// TIA Portal V19 export
FUNCTION_BLOCK "F_Zone13_FB"   // FB184, F_LAD
TITLE = SAFETY ZONE 11 - AREA 02 (FINAL CUT)
// -
// stored: Access Published
   VAR
      D14 : "Door_FB";
      D15 : "Door_FB";
      D30 : "Door_FB";
      FNS : "ForceNormalStop";
      F_SafetyValve_FinalCut { ExternalAccessible := 'False'; ExternalVisible := 'False'; ExternalWritable := 'False'} : "FDevice_Valve_FB";
      F_Contactor_HU_FinalCut_Motor { ExternalAccessible := 'False'; ExternalVisible := 'False'; ExternalWritable := 'False'} : "FDevice_Contactor_FB";
      F_Sinamics_FAK_Pusher { ExternalAccessible := 'False'; ExternalVisible := 'False'; ExternalWritable := 'False'} : "FDevice_Sinamics_FB";
      F_Sinamics_Carriage { ExternalAccessible := 'False'; ExternalVisible := 'False'; ExternalWritable := 'False'} : "FDevice_Sinamics_FB";
   END_VAR
   VAR_TEMP
      DoorNormalStop : Bool;
      DoorSafeStop : Bool;
      Door_Ok : Bool;
      DEGAS_FBK : Bool;
   END_VAR
   VAR CONSTANT
      FAK_PUSHER_S120_STOPPING_TIME : Time := T#1s;
   END_VAR
BEGIN

REGION Network 1: < < < < < < < < < < DOOR > > > > > > > > > >
END_REGION

REGION Network 2: Zone Entry enable
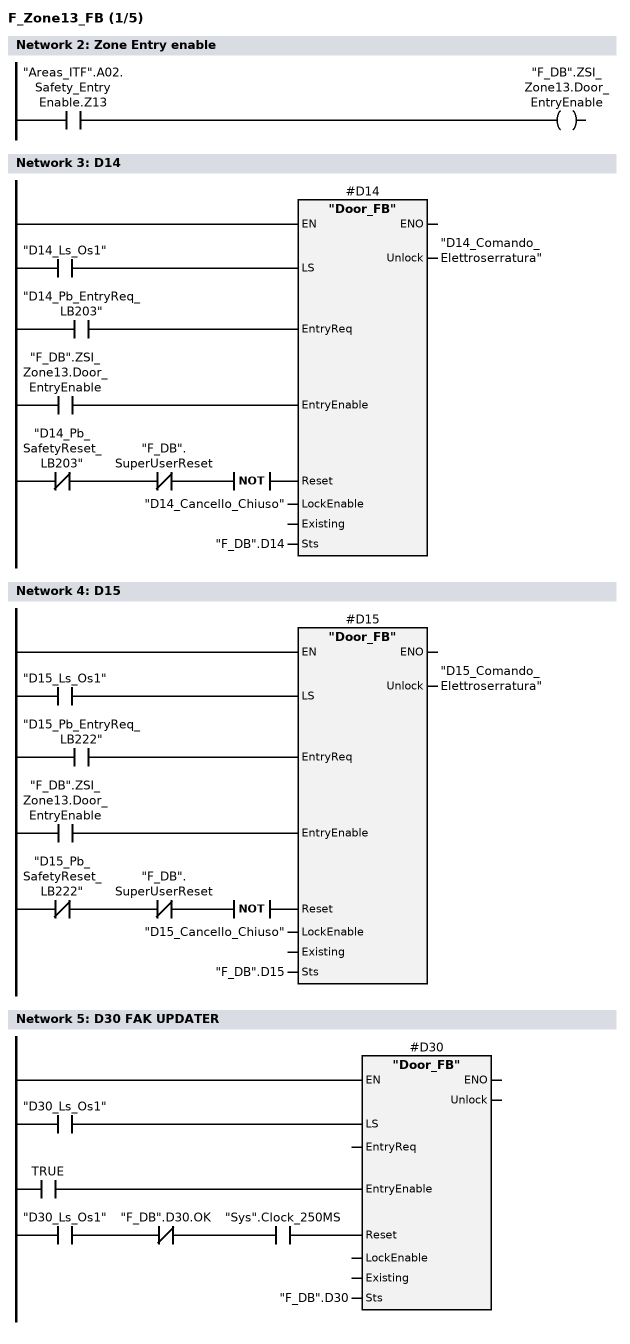
   RUNG wire#powerrail
      Contact( "Areas_ITF".A02.Safety_EntryEnable.Z13 )
      Coil( "F_DB".ZSI_Zone13.Door_EntryEnable )
   END_RUNG
   // the same network as SCL:
   "F_DB".ZSI_Zone13.Door_EntryEnable := "Areas_ITF".A02.Safety_EntryEnable.Z13;
END_REGION

REGION Network 3: D14
   RUNG wire#powerrail
      #D14(LS := wire#w1, EntryReq := wire#w2, EntryEnable := wire#w3, Reset := wire#w4, LockEnable := "D14_Cancello_Chiuso", Existing :=, Sts := "F_DB".D14, Unlock => "D14_Comando_Elettroserratura")
   END_RUNG
   RUNG wire#powerrail
      Contact( "D14_Ls_Os1" )
   END_RUNG wire#w1
   RUNG wire#powerrail
      Contact( "D14_Pb_EntryReq_LB203" )
   END_RUNG wire#w2
   RUNG wire#powerrail
      Contact( "F_DB".ZSI_Zone13.Door_EntryEnable )
   END_RUNG wire#w3
   RUNG wire#powerrail
      I_Contact( "D14_Pb_SafetyReset_LB203" )
      I_Contact( "F_DB".SuperUserReset )
      Not()
   END_RUNG wire#w4
   // the same network as SCL:
   #D14(LS := "D14_Ls_Os1",   // "Door_FB"
        EntryReq := "D14_Pb_EntryReq_LB203",
        EntryEnable := "F_DB".ZSI_Zone13.Door_EntryEnable,
        Reset := NOT (NOT "D14_Pb_SafetyReset_LB203" AND NOT "F_DB".SuperUserReset),
        LockEnable := "D14_Cancello_Chiuso",
        Sts := "F_DB".D14,
        Unlock => "D14_Comando_Elettroserratura");
END_REGION

REGION Network 4: D15
   RUNG wire#powerrail
      #D15(LS := wire#w1, EntryReq := wire#w2, EntryEnable := wire#w3, Reset := wire#w4, LockEnable := "D15_Cancello_Chiuso", Existing :=, Sts := "F_DB".D15, Unlock => "D15_Comando_Elettroserratura")
   END_RUNG
   RUNG wire#powerrail
      Contact( "D15_Ls_Os1" )
   END_RUNG wire#w1
   RUNG wire#powerrail
      Contact( "D15_Pb_EntryReq_LB222" )
   END_RUNG wire#w2
   RUNG wire#powerrail
      Contact( "F_DB".ZSI_Zone13.Door_EntryEnable )
   END_RUNG wire#w3
   RUNG wire#powerrail
      I_Contact( "D15_Pb_SafetyReset_LB222" )
      I_Contact( "F_DB".SuperUserReset )
      Not()
   END_RUNG wire#w4
   // the same network as SCL:
   #D15(LS := "D15_Ls_Os1",   // "Door_FB"
        EntryReq := "D15_Pb_EntryReq_LB222",
        EntryEnable := "F_DB".ZSI_Zone13.Door_EntryEnable,
        Reset := NOT (NOT "D15_Pb_SafetyReset_LB222" AND NOT "F_DB".SuperUserReset),
        LockEnable := "D15_Cancello_Chiuso",
        Sts := "F_DB".D15,
        Unlock => "D15_Comando_Elettroserratura");
END_REGION

REGION Network 5: D30 FAK UPDATER
   RUNG wire#powerrail
      #D30(LS := wire#w1, EntryEnable := wire#w2, Reset := wire#w3, EntryReq :=, LockEnable :=, Existing :=, Sts := "F_DB".D30, Unlock =>)
   END_RUNG
   RUNG wire#powerrail
      Contact( "D30_Ls_Os1" )
   END_RUNG wire#w1
   RUNG wire#powerrail
      Contact( TRUE )
   END_RUNG wire#w2
   RUNG wire#powerrail
      Contact( "D30_Ls_Os1" )
      I_Contact( "F_DB".D30.OK )
      Contact( "Sys".Clock_250MS )
   END_RUNG wire#w3
   // the same network as SCL:
   #D30(LS := "D30_Ls_Os1",   // "Door_FB"
        EntryEnable := TRUE,
        Reset := "D30_Ls_Os1" AND NOT "F_DB".D30.OK AND "Sys".Clock_250MS,
        Sts := "F_DB".D30);
END_REGION

REGION Network 6: < < < < < < < < < < ZONE SAFETY INTERFACE > > > > > > > > > >
END_REGION

REGION Network 7: Cumulative Zone Safety (collect)
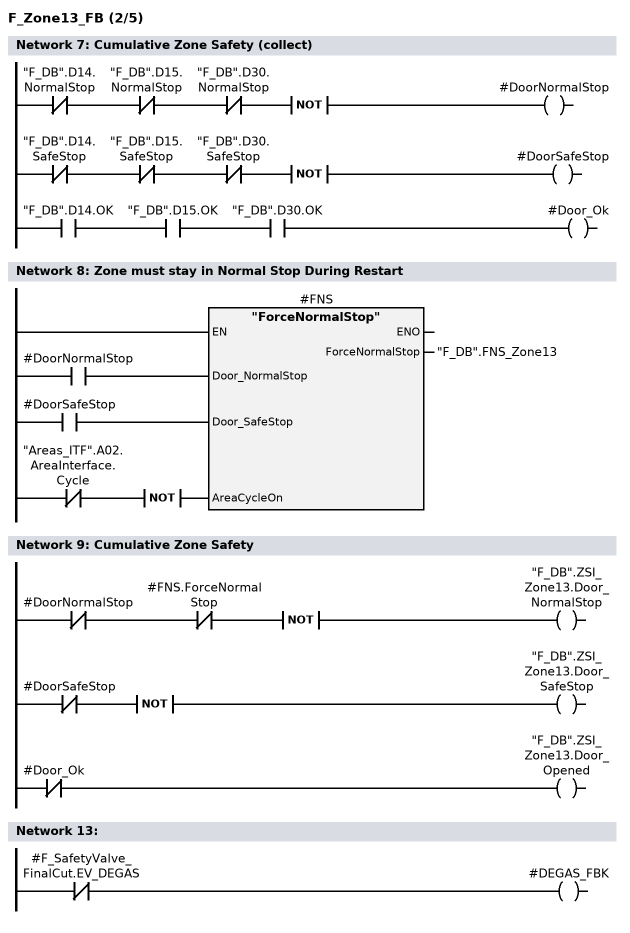
   RUNG wire#powerrail
      I_Contact( "F_DB".D14.NormalStop )
      I_Contact( "F_DB".D15.NormalStop )
      I_Contact( "F_DB".D30.NormalStop )
      Not()
      Coil( #DoorNormalStop )
   END_RUNG
   RUNG wire#powerrail
      I_Contact( "F_DB".D14.SafeStop )
      I_Contact( "F_DB".D15.SafeStop )
      I_Contact( "F_DB".D30.SafeStop )
      Not()
      Coil( #DoorSafeStop )
   END_RUNG
   RUNG wire#powerrail
      Contact( "F_DB".D14.OK )
      Contact( "F_DB".D15.OK )
      Contact( "F_DB".D30.OK )
      Coil( #Door_Ok )
   END_RUNG
   // the same network as SCL:
   #DoorNormalStop := NOT (NOT "F_DB".D14.NormalStop AND NOT "F_DB".D15.NormalStop AND NOT "F_DB".D30.NormalStop);
   #DoorSafeStop := NOT (NOT "F_DB".D14.SafeStop AND NOT "F_DB".D15.SafeStop AND NOT "F_DB".D30.SafeStop);
   #Door_Ok := "F_DB".D14.OK AND "F_DB".D15.OK AND "F_DB".D30.OK;
END_REGION

REGION Network 8: Zone must stay in Normal Stop During Restart
   RUNG wire#powerrail
      #FNS(Door_NormalStop := wire#w1, Door_SafeStop := wire#w2, AreaCycleOn := wire#w3, ForceNormalStop => "F_DB".FNS_Zone13)
   END_RUNG
   RUNG wire#powerrail
      Contact( #DoorNormalStop )
   END_RUNG wire#w1
   RUNG wire#powerrail
      Contact( #DoorSafeStop )
   END_RUNG wire#w2
   RUNG wire#powerrail
      I_Contact( "Areas_ITF".A02.AreaInterface.Cycle )
      Not()
   END_RUNG wire#w3
   // the same network as SCL:
   #FNS(Door_NormalStop := #DoorNormalStop,   // "ForceNormalStop"
        Door_SafeStop := #DoorSafeStop,
        AreaCycleOn := NOT (NOT "Areas_ITF".A02.AreaInterface.Cycle),
        ForceNormalStop => "F_DB".FNS_Zone13);
END_REGION

REGION Network 9: Cumulative Zone Safety
   RUNG wire#powerrail
      I_Contact( #DoorNormalStop )
      I_Contact( #FNS.ForceNormalStop )
      Not()
      Coil( "F_DB".ZSI_Zone13.Door_NormalStop )
   END_RUNG
   RUNG wire#powerrail
      I_Contact( #DoorSafeStop )
      Not()
      Coil( "F_DB".ZSI_Zone13.Door_SafeStop )
   END_RUNG
   RUNG wire#powerrail
      I_Contact( #Door_Ok )
      Coil( "F_DB".ZSI_Zone13.Door_Opened )
   END_RUNG
   // the same network as SCL:
   "F_DB".ZSI_Zone13.Door_NormalStop := NOT (NOT #DoorNormalStop AND NOT #FNS.ForceNormalStop);
   "F_DB".ZSI_Zone13.Door_SafeStop := NOT (NOT #DoorSafeStop);
   "F_DB".ZSI_Zone13.Door_Opened := NOT #Door_Ok;
END_REGION

REGION Network 10: >
END_REGION

REGION Network 11: >
END_REGION

REGION Network 12: < < < < < < < < < < DEVICES SAFETY VALVES > > > > > > > > > >
END_REGION

REGION Network 13
   RUNG wire#powerrail
      I_Contact( #F_SafetyValve_FinalCut.EV_DEGAS )
      Coil( #DEGAS_FBK )
   END_RUNG
   // the same network as SCL:
   #DEGAS_FBK := NOT #F_SafetyValve_FinalCut.EV_DEGAS;
END_REGION

REGION Network 14: HU A01 Safety Valve FinalCut
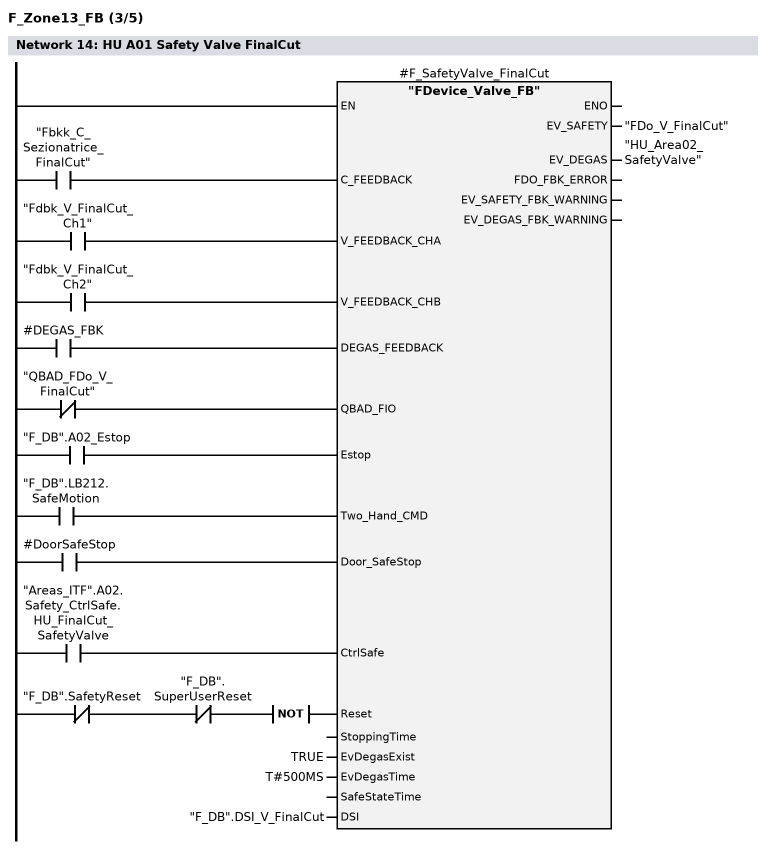
   RUNG wire#powerrail
      #F_SafetyValve_FinalCut(C_FEEDBACK := wire#w1, V_FEEDBACK_CHA := wire#w2, V_FEEDBACK_CHB := wire#w3, DEGAS_FEEDBACK := wire#w4, QBAD_FIO := wire#w5, Estop := wire#w6, Two_Hand_CMD := wire#w7, Door_SafeStop := wire#w8, CtrlSafe := wire#w9, Reset := wire#w10, StoppingTime :=, EvDegasExist := TRUE, EvDegasTime := T#500MS, SafeStateTime :=, DSI := "F_DB".DSI_V_FinalCut, EV_SAFETY => "FDo_V_FinalCut", EV_DEGAS => "HU_Area02_SafetyValve", FDO_FBK_ERROR =>, EV_SAFETY_FBK_WARNING =>, EV_DEGAS_FBK_WARNING =>)
   END_RUNG
   RUNG wire#powerrail
      Contact( "Fbkk_C_Sezionatrice_FinalCut" )
   END_RUNG wire#w1
   RUNG wire#powerrail
      Contact( "Fdbk_V_FinalCut_Ch1" )
   END_RUNG wire#w2
   RUNG wire#powerrail
      Contact( "Fdbk_V_FinalCut_Ch2" )
   END_RUNG wire#w3
   RUNG wire#powerrail
      Contact( #DEGAS_FBK )
   END_RUNG wire#w4
   RUNG wire#powerrail
      I_Contact( "QBAD_FDo_V_FinalCut" )
   END_RUNG wire#w5
   RUNG wire#powerrail
      Contact( "F_DB".A02_Estop )
   END_RUNG wire#w6
   RUNG wire#powerrail
      Contact( "F_DB".LB212.SafeMotion )
   END_RUNG wire#w7
   RUNG wire#powerrail
      Contact( #DoorSafeStop )
   END_RUNG wire#w8
   RUNG wire#powerrail
      Contact( "Areas_ITF".A02.Safety_CtrlSafe.HU_FinalCut_SafetyValve )
   END_RUNG wire#w9
   RUNG wire#powerrail
      I_Contact( "F_DB".SafetyReset )
      I_Contact( "F_DB".SuperUserReset )
      Not()
   END_RUNG wire#w10
   // the same network as SCL:
   #F_SafetyValve_FinalCut(C_FEEDBACK := "Fbkk_C_Sezionatrice_FinalCut",   // "FDevice_Valve_FB"
                           V_FEEDBACK_CHA := "Fdbk_V_FinalCut_Ch1",
                           V_FEEDBACK_CHB := "Fdbk_V_FinalCut_Ch2",
                           DEGAS_FEEDBACK := #DEGAS_FBK,
                           QBAD_FIO := NOT "QBAD_FDo_V_FinalCut",
                           Estop := "F_DB".A02_Estop,
                           Two_Hand_CMD := "F_DB".LB212.SafeMotion,
                           Door_SafeStop := #DoorSafeStop,
                           CtrlSafe := "Areas_ITF".A02.Safety_CtrlSafe.HU_FinalCut_SafetyValve,
                           Reset := NOT (NOT "F_DB".SafetyReset AND NOT "F_DB".SuperUserReset),
                           EvDegasExist := TRUE,
                           EvDegasTime := T#500MS,
                           DSI := "F_DB".DSI_V_FinalCut,
                           EV_SAFETY => "FDo_V_FinalCut",
                           EV_DEGAS => "HU_Area02_SafetyValve");
END_REGION

REGION Network 15: >
END_REGION

REGION Network 16: >
END_REGION

REGION Network 17: < < < < < < < < < < DEVICES CONTACTORS > > > > > > > > > >
END_REGION

REGION Network 18: HU Final cut Motor contactor
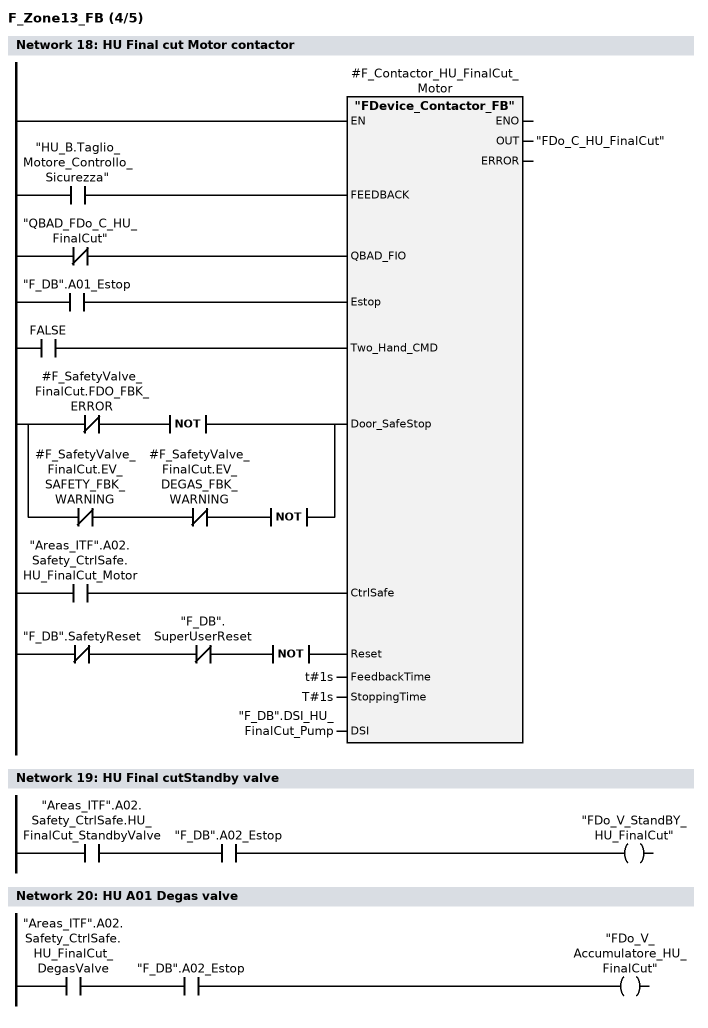
   RUNG wire#powerrail
      #F_Contactor_HU_FinalCut_Motor(FEEDBACK := wire#w1, QBAD_FIO := wire#w2, Estop := wire#w3, Two_Hand_CMD := wire#w4, Door_SafeStop := wire#w5, CtrlSafe := wire#w6, Reset := wire#w7, FeedbackTime := t#1s, StoppingTime := T#1s, DSI := "F_DB".DSI_HU_FinalCut_Pump, OUT => "FDo_C_HU_FinalCut", ERROR =>)
   END_RUNG
   RUNG wire#powerrail
      Contact( "HU_B.Taglio_Motore_Controllo_Sicurezza" )
   END_RUNG wire#w1
   RUNG wire#powerrail
      I_Contact( "QBAD_FDo_C_HU_FinalCut" )
   END_RUNG wire#w2
   RUNG wire#powerrail
      Contact( "F_DB".A01_Estop )
   END_RUNG wire#w3
   RUNG wire#powerrail
      Contact( FALSE )
   END_RUNG wire#w4
   RUNG wire#powerrail
      I_Contact( #F_SafetyValve_FinalCut.FDO_FBK_ERROR )
      Not()
   END_RUNG wire#w5
   RUNG wire#powerrail
      I_Contact( #F_SafetyValve_FinalCut.EV_SAFETY_FBK_WARNING )
      I_Contact( #F_SafetyValve_FinalCut.EV_DEGAS_FBK_WARNING )
      Not()
   END_RUNG wire#w5
   RUNG wire#powerrail
      Contact( "Areas_ITF".A02.Safety_CtrlSafe.HU_FinalCut_Motor )
   END_RUNG wire#w6
   RUNG wire#powerrail
      I_Contact( "F_DB".SafetyReset )
      I_Contact( "F_DB".SuperUserReset )
      Not()
   END_RUNG wire#w7
   // the same network as SCL:
   #F_Contactor_HU_FinalCut_Motor(FEEDBACK := "HU_B.Taglio_Motore_Controllo_Sicurezza",   // "FDevice_Contactor_FB"
                           QBAD_FIO := NOT "QBAD_FDo_C_HU_FinalCut",
                           Estop := "F_DB".A01_Estop,
                           Two_Hand_CMD := FALSE,
                           Door_SafeStop := NOT (NOT #F_SafetyValve_FinalCut.FDO_FBK_ERROR) OR NOT (NOT #F_SafetyValve_FinalCut.EV_SAFETY_FBK_WARNING AND NOT #F_SafetyValve_FinalCut.EV_DEGAS_FBK_WARNING),
                           CtrlSafe := "Areas_ITF".A02.Safety_CtrlSafe.HU_FinalCut_Motor,
                           Reset := NOT (NOT "F_DB".SafetyReset AND NOT "F_DB".SuperUserReset),
                           FeedbackTime := t#1s,
                           StoppingTime := T#1s,
                           DSI := "F_DB".DSI_HU_FinalCut_Pump,
                           OUT => "FDo_C_HU_FinalCut");
END_REGION

REGION Network 19: HU Final cutStandby valve
   RUNG wire#powerrail
      Contact( "Areas_ITF".A02.Safety_CtrlSafe.HU_FinalCut_StandbyValve )
      Contact( "F_DB".A02_Estop )
      Coil( "FDo_V_StandBY_HU_FinalCut" )
   END_RUNG
   // the same network as SCL:
   "FDo_V_StandBY_HU_FinalCut" := "Areas_ITF".A02.Safety_CtrlSafe.HU_FinalCut_StandbyValve AND "F_DB".A02_Estop;
END_REGION

REGION Network 20: HU A01 Degas valve
   RUNG wire#powerrail
      Contact( "Areas_ITF".A02.Safety_CtrlSafe.HU_FinalCut_DegasValve )
      Contact( "F_DB".A02_Estop )
      Coil( "FDo_V_Accumulatore_HU_FinalCut" )
   END_RUNG
   // the same network as SCL:
   "FDo_V_Accumulatore_HU_FinalCut" := "Areas_ITF".A02.Safety_CtrlSafe.HU_FinalCut_DegasValve AND "F_DB".A02_Estop;
END_REGION

REGION Network 21: >
END_REGION

REGION Network 22: >
END_REGION

REGION Network 23: < < < < < < < < < < DEVICES S120 > > > > > > > > > >
END_REGION

REGION Network 24: S120 - FAK Pusher Ax
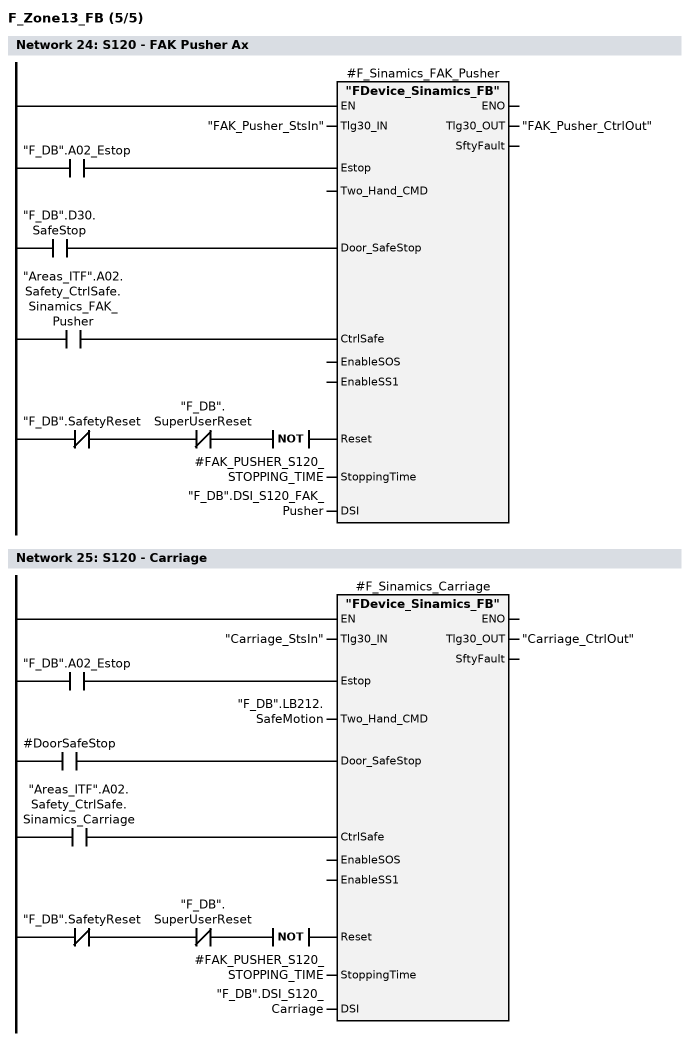
   RUNG wire#powerrail
      #F_Sinamics_FAK_Pusher(Estop := wire#w1, Door_SafeStop := wire#w2, CtrlSafe := wire#w3, Reset := wire#w4, Tlg30_IN := "FAK_Pusher_StsIn", Two_Hand_CMD :=, EnableSOS :=, EnableSS1 :=, StoppingTime := #FAK_PUSHER_S120_STOPPING_TIME, DSI := "F_DB".DSI_S120_FAK_Pusher, Tlg30_OUT => "FAK_Pusher_CtrlOut", SftyFault =>)
   END_RUNG
   RUNG wire#powerrail
      Contact( "F_DB".A02_Estop )
   END_RUNG wire#w1
   RUNG wire#powerrail
      Contact( "F_DB".D30.SafeStop )
   END_RUNG wire#w2
   RUNG wire#powerrail
      Contact( "Areas_ITF".A02.Safety_CtrlSafe.Sinamics_FAK_Pusher )
   END_RUNG wire#w3
   RUNG wire#powerrail
      I_Contact( "F_DB".SafetyReset )
      I_Contact( "F_DB".SuperUserReset )
      Not()
   END_RUNG wire#w4
   // the same network as SCL:
   #F_Sinamics_FAK_Pusher(Tlg30_IN := "FAK_Pusher_StsIn",   // "FDevice_Sinamics_FB"
                          Estop := "F_DB".A02_Estop,
                          Door_SafeStop := "F_DB".D30.SafeStop,
                          CtrlSafe := "Areas_ITF".A02.Safety_CtrlSafe.Sinamics_FAK_Pusher,
                          Reset := NOT (NOT "F_DB".SafetyReset AND NOT "F_DB".SuperUserReset),
                          StoppingTime := #FAK_PUSHER_S120_STOPPING_TIME,
                          DSI := "F_DB".DSI_S120_FAK_Pusher,
                          Tlg30_OUT => "FAK_Pusher_CtrlOut");
END_REGION

REGION Network 25: S120 - Carriage
   RUNG wire#powerrail
      #F_Sinamics_Carriage(Estop := wire#w1, Door_SafeStop := wire#w2, CtrlSafe := wire#w3, Reset := wire#w4, Tlg30_IN := "Carriage_StsIn", Two_Hand_CMD := "F_DB".LB212.SafeMotion, EnableSOS :=, EnableSS1 :=, StoppingTime := #FAK_PUSHER_S120_STOPPING_TIME, DSI := "F_DB".DSI_S120_Carriage, Tlg30_OUT => "Carriage_CtrlOut", SftyFault =>)
   END_RUNG
   RUNG wire#powerrail
      Contact( "F_DB".A02_Estop )
   END_RUNG wire#w1
   RUNG wire#powerrail
      Contact( #DoorSafeStop )
   END_RUNG wire#w2
   RUNG wire#powerrail
      Contact( "Areas_ITF".A02.Safety_CtrlSafe.Sinamics_Carriage )
   END_RUNG wire#w3
   RUNG wire#powerrail
      I_Contact( "F_DB".SafetyReset )
      I_Contact( "F_DB".SuperUserReset )
      Not()
   END_RUNG wire#w4
   // the same network as SCL:
   #F_Sinamics_Carriage(Tlg30_IN := "Carriage_StsIn",   // "FDevice_Sinamics_FB"
                        Estop := "F_DB".A02_Estop,
                        Two_Hand_CMD := "F_DB".LB212.SafeMotion,
                        Door_SafeStop := #DoorSafeStop,
                        CtrlSafe := "Areas_ITF".A02.Safety_CtrlSafe.Sinamics_Carriage,
                        Reset := NOT (NOT "F_DB".SafetyReset AND NOT "F_DB".SuperUserReset),
                        StoppingTime := #FAK_PUSHER_S120_STOPPING_TIME,
                        DSI := "F_DB".DSI_S120_Carriage,
                        Tlg30_OUT => "Carriage_CtrlOut");
END_REGION

REGION Network 26: >
END_REGION

REGION Network 27: >
END_REGION
END_FUNCTION_BLOCK
